FUNCTION GetBit : BOOL
VAR_INPUT
	Value: ULINT;
	BitNr: INT;
END_VAR
VAR
END_VAR

GetBit := (Value AND SHL(INT_TO_ULINT(1), BitNr)) <> 0;

END_FUNCTION

(* stored: Version 1.1.0.1, ProductVersion 3.1.4024.3
   POU GetBit: Id {a698304e-48d3-4e0e-b267-b99a1011644f}, SpecialFunc None *)
